   // // TIF[14].SBottom : Werkeug neu: Größe unten / Tool new: size bottom / Herramienta nueva: tamaño abajo
   // // TIF[15].SBottom : Werkeug neu: Größe unten / Tool new: size bottom / Herramienta nueva: tamaño abajo
   // // TIF[16].SBottom : Werkeug neu: Größe unten / Tool new: size bottom / Herramienta nueva: tamaño abajo
   // // TIF[2].TInBuffer : ID für Werkzeuge im Puffer / ID for tools in buffer / ID para herramientas en búfer
   // // TIF[3].TInBuffer : ID für Werkzeuge im Puffer / ID for tools in buffer / ID para herramientas en búfer
   // // TIF[4].TInBuffer : ID für Werkzeuge im Puffer / ID for tools in buffer / ID para herramientas en búfer
   // // TIF[5].TInBuffer : ID für Werkzeuge im Puffer / ID for tools in buffer / ID para herramientas en búfer
   // // TIF[6].TInBuffer : ID für Werkzeuge im Puffer / ID for tools in buffer / ID para herramientas en búfer
   // // TIF[7].TInBuffer : ID für Werkzeuge im Puffer / ID for tools in buffer / ID para herramientas en búfer
   // // TIF[8].TInBuffer : ID für Werkzeuge im Puffer / ID for tools in buffer / ID para herramientas en búfer
   // // TIF[9].TInBuffer : ID für Werkzeuge im Puffer / ID for tools in buffer / ID para herramientas en búfer
   // // TIF[10].TInBuffer : ID für Werkzeuge im Puffer / ID for tools in buffer / ID para herramientas en búfer
   // // TIF[11].TInBuffer : ID für Werkzeuge im Puffer / ID for tools in buffer / ID para herramientas en búfer
   // // TIF[12].TInBuffer : ID für Werkzeuge im Puffer / ID for tools in buffer / ID para herramientas en búfer
   // // TIF[13].TInBuffer : ID für Werkzeuge im Puffer / ID for tools in buffer / ID para herramientas en búfer
   // // TIF[14].TInBuffer : ID für Werkzeuge im Puffer / ID for tools in buffer / ID para herramientas en búfer
   // // TIF[15].TInBuffer : ID für Werkzeuge im Puffer / ID for tools in buffer / ID para herramientas en búfer
   // // TIF[16].TInBuffer : ID für Werkzeuge im Puffer / ID for tools in buffer / ID para herramientas en búfer
   // // TIF[2].IgnoreDisabled : Deaktiviert ignorieren / Ignore disabled / Ignorar desactivado
   // // TIF[3].IgnoreDisabled : Deaktiviert ignorieren / Ignore disabled / Ignorar desactivado
   // // TIF[4].IgnoreDisabled : Deaktiviert ignorieren / Ignore disabled / Ignorar desactivado
   // // TIF[5].IgnoreDisabled : Deaktiviert ignorieren / Ignore disabled / Ignorar desactivado
   // // TIF[6].IgnoreDisabled : Deaktiviert ignorieren / Ignore disabled / Ignorar desactivado
   // // TIF[7].IgnoreDisabled : Deaktiviert ignorieren / Ignore disabled / Ignorar desactivado
   // // TIF[8].IgnoreDisabled : Deaktiviert ignorieren / Ignore disabled / Ignorar desactivado
   // // TIF[9].IgnoreDisabled : Deaktiviert ignorieren / Ignore disabled / Ignorar desactivado
   // // TIF[10].IgnoreDisabled : Deaktiviert ignorieren / Ignore disabled / Ignorar desactivado
   // // TIF[11].IgnoreDisabled : Deaktiviert ignorieren / Ignore disabled / Ignorar desactivado
   // // TIF[12].IgnoreDisabled : Deaktiviert ignorieren / Ignore disabled / Ignorar desactivado
   // // TIF[13].IgnoreDisabled : Deaktiviert ignorieren / Ignore disabled / Ignorar desactivado
   // // TIF[14].IgnoreDisabled : Deaktiviert ignorieren / Ignore disabled / Ignorar desactivado
   // // TIF[15].IgnoreDisabled : Deaktiviert ignorieren / Ignore disabled / Ignorar desactivado
   // // TIF[16].IgnoreDisabled : Deaktiviert ignorieren / Ignore disabled / Ignorar desactivado
   // // TIF[2].Unload : Zu entladen / To be unloaded / Por descargar
   // // TIF[3].Unload : Zu entladen / To be unloaded / Por descargar
   // // TIF[4].Unload : Zu entladen / To be unloaded / Por descargar
   // // TIF[5].Unload : Zu entladen / To be unloaded / Por descargar
   // // TIF[6].Unload : Zu entladen / To be unloaded / Por descargar
   // // TIF[7].Unload : Zu entladen / To be unloaded / Por descargar
   // // TIF[8].Unload : Zu entladen / To be unloaded / Por descargar
   // // TIF[9].Unload : Zu entladen / To be unloaded / Por descargar
   // // TIF[10].Unload : Zu entladen / To be unloaded / Por descargar
   // // TIF[11].Unload : Zu entladen / To be unloaded / Por descargar
   // // TIF[12].Unload : Zu entladen / To be unloaded / Por descargar
   // // TIF[13].Unload : Zu entladen / To be unloaded / Por descargar
   // // TIF[14].Unload : Zu entladen / To be unloaded / Por descargar
   // // TIF[15].Unload : Zu entladen / To be unloaded / Por descargar
   // // TIF[16].Unload : Zu entladen / To be unloaded / Por descargar
   // // TIF[2].Load : Zu laden / To be loaded / Por cargar
   // // TIF[3].Load : Zu laden / To be loaded / Por cargar
   // // TIF[4].Load : Zu laden / To be loaded / Por cargar
   // // TIF[5].Load : Zu laden / To be loaded / Por cargar
   // // TIF[6].Load : Zu laden / To be loaded / Por cargar
   // // TIF[7].Load : Zu laden / To be loaded / Por cargar
   // // TIF[8].Load : Zu laden / To be loaded / Por cargar
   // // TIF[9].Load : Zu laden / To be loaded / Por cargar
   // // TIF[10].Load : Zu laden / To be loaded / Por cargar
   // // TIF[11].Load : Zu laden / To be loaded / Por cargar
   // // TIF[12].Load : Zu laden / To be loaded / Por cargar
   // // TIF[13].Load : Zu laden / To be loaded / Por cargar
   // // TIF[14].Load : Zu laden / To be loaded / Por cargar
   // // TIF[15].Load : Zu laden / To be loaded / Por cargar
   // // TIF[16].Load : Zu laden / To be loaded / Por cargar
   // // TIF[2].MasterTool : Master-Werkzeug / Master tool / Herramienta maestra
   // // TIF[3].MasterTool : Master-Werkzeug / Master tool / Herramienta maestra
   // // TIF[4].MasterTool : Master-Werkzeug / Master tool / Herramienta maestra
   // // TIF[5].MasterTool : Master-Werkzeug / Master tool / Herramienta maestra
   // // TIF[6].MasterTool : Master-Werkzeug / Master tool / Herramienta maestra
   // // TIF[7].MasterTool : Master-Werkzeug / Master tool / Herramienta maestra
   // // TIF[8].MasterTool : Master-Werkzeug / Master tool / Herramienta maestra
   // // TIF[9].MasterTool : Master-Werkzeug / Master tool / Herramienta maestra
   // // TIF[10].MasterTool : Master-Werkzeug / Master tool / Herramienta maestra
   // // TIF[11].MasterTool : Master-Werkzeug / Master tool / Herramienta maestra
   // // TIF[12].MasterTool : Master-Werkzeug / Master tool / Herramienta maestra
   // // TIF[13].MasterTool : Master-Werkzeug / Master tool / Herramienta maestra
   // // TIF[14].MasterTool : Master-Werkzeug / Master tool / Herramienta maestra
   // // TIF[15].MasterTool : Master-Werkzeug / Master tool / Herramienta maestra
   // // TIF[16].MasterTool : Master-Werkzeug / Master tool / Herramienta maestra
   // // TIF[2].n38_5 : Reserviert / Reserved / Reservado
   // // TIF[3].n38_5 : Reserviert / Reserved / Reservado
   // // TIF[4].n38_5 : Reserviert / Reserved / Reservado
   // // TIF[5].n38_5 : Reserviert / Reserved / Reservado
   // // TIF[6].n38_5 : Reserviert / Reserved / Reservado
   // // TIF[7].n38_5 : Reserviert / Reserved / Reservado
   // // TIF[8].n38_5 : Reserviert / Reserved / Reservado
   // // TIF[9].n38_5 : Reserviert / Reserved / Reservado
   // // TIF[10].n38_5 : Reserviert / Reserved / Reservado
   // // TIF[11].n38_5 : Reserviert / Reserved / Reservado
   // // TIF[12].n38_5 : Reserviert / Reserved / Reservado
   // // TIF[13].n38_5 : Reserviert / Reserved / Reservado
   // // TIF[14].n38_5 : Reserviert / Reserved / Reservado
   // // TIF[15].n38_5 : Reserviert / Reserved / Reservado
   // // TIF[16].n38_5 : Reserviert / Reserved / Reservado
   // // TIF[2].Exchange_1to1 : 1:1 Austausch / 1:1 exchange / Cambio 1:1
   // // TIF[3].Exchange_1to1 : 1:1 Austausch / 1:1 exchange / Cambio 1:1
   // // TIF[4].Exchange_1to1 : 1:1 Austausch / 1:1 exchange / Cambio 1:1
   // // TIF[5].Exchange_1to1 : 1:1 Austausch / 1:1 exchange / Cambio 1:1
   // // TIF[6].Exchange_1to1 : 1:1 Austausch / 1:1 exchange / Cambio 1:1
   // // TIF[7].Exchange_1to1 : 1:1 Austausch / 1:1 exchange / Cambio 1:1
   // // TIF[8].Exchange_1to1 : 1:1 Austausch / 1:1 exchange / Cambio 1:1
   // // TIF[9].Exchange_1to1 : 1:1 Austausch / 1:1 exchange / Cambio 1:1
   // // TIF[10].Exchange_1to1 : 1:1 Austausch / 1:1 exchange / Cambio 1:1
   // // TIF[11].Exchange_1to1 : 1:1 Austausch / 1:1 exchange / Cambio 1:1
   // // TIF[12].Exchange_1to1 : 1:1 Austausch / 1:1 exchange / Cambio 1:1
   // // TIF[13].Exchange_1to1 : 1:1 Austausch / 1:1 exchange / Cambio 1:1
   // // TIF[14].Exchange_1to1 : 1:1 Austausch / 1:1 exchange / Cambio 1:1
   // // TIF[15].Exchange_1to1 : 1:1 Austausch / 1:1 exchange / Cambio 1:1
   // // TIF[16].Exchange_1to1 : 1:1 Austausch / 1:1 exchange / Cambio 1:1
   // // TIF[2].HandTool : Handwerkzeug / Hand tool / Herramienta manual
   // // TIF[3].HandTool : Handwerkzeug / Hand tool / Herramienta manual
   // // TIF[4].HandTool : Handwerkzeug / Hand tool / Herramienta manual
   // // TIF[5].HandTool : Handwerkzeug / Hand tool / Herramienta manual
   // // TIF[6].HandTool : Handwerkzeug / Hand tool / Herramienta manual
   // // TIF[7].HandTool : Handwerkzeug / Hand tool / Herramienta manual
   // // TIF[8].HandTool : Handwerkzeug / Hand tool / Herramienta manual
   // // TIF[9].HandTool : Handwerkzeug / Hand tool / Herramienta manual
   // // TIF[10].HandTool : Handwerkzeug / Hand tool / Herramienta manual
   // // TIF[11].HandTool : Handwerkzeug / Hand tool / Herramienta manual
   // // TIF[12].HandTool : Handwerkzeug / Hand tool / Herramienta manual
   // // TIF[13].HandTool : Handwerkzeug / Hand tool / Herramienta manual
   // // TIF[14].HandTool : Handwerkzeug / Hand tool / Herramienta manual
   // // TIF[15].HandTool : Handwerkzeug / Hand tool / Herramienta manual
   // // TIF[16].HandTool : Handwerkzeug / Hand tool / Herramienta manual
   // // TIF[2].Active : Aktives Werkzeug / Active tool / Herramienta activa
   // // TIF[3].Active : Aktives Werkzeug / Active tool / Herramienta activa
   // // TIF[4].Active : Aktives Werkzeug / Active tool / Herramienta activa
   // // TIF[5].Active : Aktives Werkzeug / Active tool / Herramienta activa
   // // TIF[6].Active : Aktives Werkzeug / Active tool / Herramienta activa
   // // TIF[7].Active : Aktives Werkzeug / Active tool / Herramienta activa
   // // TIF[8].Active : Aktives Werkzeug / Active tool / Herramienta activa
   // // TIF[9].Active : Aktives Werkzeug / Active tool / Herramienta activa
   // // TIF[10].Active : Aktives Werkzeug / Active tool / Herramienta activa
   // // TIF[11].Active : Aktives Werkzeug / Active tool / Herramienta activa
   // // TIF[12].Active : Aktives Werkzeug / Active tool / Herramienta activa
   // // TIF[13].Active : Aktives Werkzeug / Active tool / Herramienta activa
   // // TIF[14].Active : Aktives Werkzeug / Active tool / Herramienta activa
   // // TIF[15].Active : Aktives Werkzeug / Active tool / Herramienta activa
   // // TIF[16].Active : Aktives Werkzeug / Active tool / Herramienta activa
   // // TIF[2].Enabled : Werkzeug aktiviert / Tool enabled / Herramienta activada
   // // TIF[3].Enabled : Werkzeug aktiviert / Tool enabled / Herramienta activada
   // // TIF[4].Enabled : Werkzeug aktiviert / Tool enabled / Herramienta activada
   // // TIF[5].Enabled : Werkzeug aktiviert / Tool enabled / Herramienta activada
   // // TIF[6].Enabled : Werkzeug aktiviert / Tool enabled / Herramienta activada
   // // TIF[7].Enabled : Werkzeug aktiviert / Tool enabled / Herramienta activada
   // // TIF[8].Enabled : Werkzeug aktiviert / Tool enabled / Herramienta activada
   // // TIF[9].Enabled : Werkzeug aktiviert / Tool enabled / Herramienta activada
   // // TIF[10].Enabled : Werkzeug aktiviert / Tool enabled / Herramienta activada
   // // TIF[11].Enabled : Werkzeug aktiviert / Tool enabled / Herramienta activada
   // // TIF[12].Enabled : Werkzeug aktiviert / Tool enabled / Herramienta activada
   // // TIF[13].Enabled : Werkzeug aktiviert / Tool enabled / Herramienta activada
   // // TIF[14].Enabled : Werkzeug aktiviert / Tool enabled / Herramienta activada
   // // TIF[15].Enabled : Werkzeug aktiviert / Tool enabled / Herramienta activada
   // // TIF[16].Enabled : Werkzeug aktiviert / Tool enabled / Herramienta activada
   // // TIF[2].Disabled : Werkzeug deaktiviert / Tool disabled / Herramienta desactivada
   // // TIF[3].Disabled : Werkzeug deaktiviert / Tool disabled / Herramienta desactivada
   // // TIF[4].Disabled : Werkzeug deaktiviert / Tool disabled / Herramienta desactivada
   // // TIF[5].Disabled : Werkzeug deaktiviert / Tool disabled / Herramienta desactivada
   // // TIF[6].Disabled : Werkzeug deaktiviert / Tool disabled / Herramienta desactivada
   // // TIF[7].Disabled : Werkzeug deaktiviert / Tool disabled / Herramienta desactivada
   // // TIF[8].Disabled : Werkzeug deaktiviert / Tool disabled / Herramienta desactivada
   // // TIF[9].Disabled : Werkzeug deaktiviert / Tool disabled / Herramienta desactivada
   // // TIF[10].Disabled : Werkzeug deaktiviert / Tool disabled / Herramienta desactivada
   // // TIF[11].Disabled : Werkzeug deaktiviert / Tool disabled / Herramienta desactivada
   // // TIF[12].Disabled : Werkzeug deaktiviert / Tool disabled / Herramienta desactivada
   // // TIF[13].Disabled : Werkzeug deaktiviert / Tool disabled / Herramienta desactivada
   // // TIF[14].Disabled : Werkzeug deaktiviert / Tool disabled / Herramienta desactivada
   // // TIF[15].Disabled : Werkzeug deaktiviert / Tool disabled / Herramienta desactivada
   // // TIF[16].Disabled : Werkzeug deaktiviert / Tool disabled / Herramienta desactivada
   // // TIF[2].Measured : Werkzeug gemessen / Tool measured / Herramienta medida
   // // TIF[3].Measured : Werkzeug gemessen / Tool measured / Herramienta medida
   // // TIF[4].Measured : Werkzeug gemessen / Tool measured / Herramienta medida
   // // TIF[5].Measured : Werkzeug gemessen / Tool measured / Herramienta medida
   // // TIF[6].Measured : Werkzeug gemessen / Tool measured / Herramienta medida
   // // TIF[7].Measured : Werkzeug gemessen / Tool measured / Herramienta medida
   // // TIF[8].Measured : Werkzeug gemessen / Tool measured / Herramienta medida
   // // TIF[9].Measured : Werkzeug gemessen / Tool measured / Herramienta medida
   // // TIF[10].Measured : Werkzeug gemessen / Tool measured / Herramienta medida
   // // TIF[11].Measured : Werkzeug gemessen / Tool measured / Herramienta medida
   // // TIF[12].Measured : Werkzeug gemessen / Tool measured / Herramienta medida
   // // TIF[13].Measured : Werkzeug gemessen / Tool measured / Herramienta medida
   // // TIF[14].Measured : Werkzeug gemessen / Tool measured / Herramienta medida
   // // TIF[15].Measured : Werkzeug gemessen / Tool measured / Herramienta medida
   // // TIF[16].Measured : Werkzeug gemessen / Tool measured / Herramienta medida
   // // TIF[2].Prewarn : Vorwarnungsgrenze erreicht / Prewarning limit reached / Límite de prealarma alcanzado
   // // TIF[3].Prewarn : Vorwarnungsgrenze erreicht / Prewarning limit reached / Límite de prealarma alcanzado
   // // TIF[4].Prewarn : Vorwarnungsgrenze erreicht / Prewarning limit reached / Límite de prealarma alcanzado
   // // TIF[5].Prewarn : Vorwarnungsgrenze erreicht / Prewarning limit reached / Límite de prealarma alcanzado
   // // TIF[6].Prewarn : Vorwarnungsgrenze erreicht / Prewarning limit reached / Límite de prealarma alcanzado
   // // TIF[7].Prewarn : Vorwarnungsgrenze erreicht / Prewarning limit reached / Límite de prealarma alcanzado
   // // TIF[8].Prewarn : Vorwarnungsgrenze erreicht / Prewarning limit reached / Límite de prealarma alcanzado
   // // TIF[9].Prewarn : Vorwarnungsgrenze erreicht / Prewarning limit reached / Límite de prealarma alcanzado
   // // TIF[10].Prewarn : Vorwarnungsgrenze erreicht / Prewarning limit reached / Límite de prealarma alcanzado
   // // TIF[11].Prewarn : Vorwarnungsgrenze erreicht / Prewarning limit reached / Límite de prealarma alcanzado
   // // TIF[12].Prewarn : Vorwarnungsgrenze erreicht / Prewarning limit reached / Límite de prealarma alcanzado
   // // TIF[13].Prewarn : Vorwarnungsgrenze erreicht / Prewarning limit reached / Límite de prealarma alcanzado
   // // TIF[14].Prewarn : Vorwarnungsgrenze erreicht / Prewarning limit reached / Límite de prealarma alcanzado
   // // TIF[15].Prewarn : Vorwarnungsgrenze erreicht / Prewarning limit reached / Límite de prealarma alcanzado
   // // TIF[16].Prewarn : Vorwarnungsgrenze erreicht / Prewarning limit reached / Límite de prealarma alcanzado
   // // TIF[2].Change : Werkzeug wird gewechselt / Tool being changed / Sustituyendo herramienta
   // // TIF[3].Change : Werkzeug wird gewechselt / Tool being changed / Sustituyendo herramienta
   // // TIF[4].Change : Werkzeug wird gewechselt / Tool being changed / Sustituyendo herramienta
   // // TIF[5].Change : Werkzeug wird gewechselt / Tool being changed / Sustituyendo herramienta
   // // TIF[6].Change : Werkzeug wird gewechselt / Tool being changed / Sustituyendo herramienta
   // // TIF[7].Change : Werkzeug wird gewechselt / Tool being changed / Sustituyendo herramienta
   // // TIF[8].Change : Werkzeug wird gewechselt / Tool being changed / Sustituyendo herramienta
   // // TIF[9].Change : Werkzeug wird gewechselt / Tool being changed / Sustituyendo herramienta
   // // TIF[10].Change : Werkzeug wird gewechselt / Tool being changed / Sustituyendo herramienta
   // // TIF[11].Change : Werkzeug wird gewechselt / Tool being changed / Sustituyendo herramienta
   // // TIF[12].Change : Werkzeug wird gewechselt / Tool being changed / Sustituyendo herramienta
   // // TIF[13].Change : Werkzeug wird gewechselt / Tool being changed / Sustituyendo herramienta
   // // TIF[14].Change : Werkzeug wird gewechselt / Tool being changed / Sustituyendo herramienta
   // // TIF[15].Change : Werkzeug wird gewechselt / Tool being changed / Sustituyendo herramienta
   // // TIF[16].Change : Werkzeug wird gewechselt / Tool being changed / Sustituyendo herramienta
   // // TIF[2].FixedLoc : Werkzeug-Festplatz codiert / Tool fixed location coded / Puesto fijo de herramienta codificado
   // // TIF[3].FixedLoc : Werkzeug-Festplatz codiert / Tool fixed location coded / Puesto fijo de herramienta codificado
   // // TIF[4].FixedLoc : Werkzeug-Festplatz codiert / Tool fixed location coded / Puesto fijo de herramienta codificado
   // // TIF[5].FixedLoc : Werkzeug-Festplatz codiert / Tool fixed location coded / Puesto fijo de herramienta codificado
   // // TIF[6].FixedLoc : Werkzeug-Festplatz codiert / Tool fixed location coded / Puesto fijo de herramienta codificado
   // // TIF[7].FixedLoc : Werkzeug-Festplatz codiert / Tool fixed location coded / Puesto fijo de herramienta codificado
   // // TIF[8].FixedLoc : Werkzeug-Festplatz codiert / Tool fixed location coded / Puesto fijo de herramienta codificado
   // // TIF[9].FixedLoc : Werkzeug-Festplatz codiert / Tool fixed location coded / Puesto fijo de herramienta codificado
   // // TIF[10].FixedLoc : Werkzeug-Festplatz codiert / Tool fixed location coded / Puesto fijo de herramienta codificado
   // // TIF[11].FixedLoc : Werkzeug-Festplatz codiert / Tool fixed location coded / Puesto fijo de herramienta codificado
   // // TIF[12].FixedLoc : Werkzeug-Festplatz codiert / Tool fixed location coded / Puesto fijo de herramienta codificado
   // // TIF[13].FixedLoc : Werkzeug-Festplatz codiert / Tool fixed location coded / Puesto fijo de herramienta codificado
   // // TIF[14].FixedLoc : Werkzeug-Festplatz codiert / Tool fixed location coded / Puesto fijo de herramienta codificado
   // // TIF[15].FixedLoc : Werkzeug-Festplatz codiert / Tool fixed location coded / Puesto fijo de herramienta codificado
   // // TIF[16].FixedLoc : Werkzeug-Festplatz codiert / Tool fixed location coded / Puesto fijo de herramienta codificado
   // // TIF[2].Used : Werkzeug war in Gebrauch / Tool was in use / La herramienta estaba en uso
   // // TIF[3].Used : Werkzeug war in Gebrauch / Tool was in use / La herramienta estaba en uso
   // // TIF[4].Used : Werkzeug war in Gebrauch / Tool was in use / La herramienta estaba en uso
   // // TIF[5].Used : Werkzeug war in Gebrauch / Tool was in use / La herramienta estaba en uso
   // // TIF[6].Used : Werkzeug war in Gebrauch / Tool was in use / La herramienta estaba en uso
   // // TIF[7].Used : Werkzeug war in Gebrauch / Tool was in use / La herramienta estaba en uso
   // // TIF[8].Used : Werkzeug war in Gebrauch / Tool was in use / La herramienta estaba en uso
   // // TIF[9].Used : Werkzeug war in Gebrauch / Tool was in use / La herramienta estaba en uso
   // // TIF[10].Used : Werkzeug war in Gebrauch / Tool was in use / La herramienta estaba en uso
   // // TIF[11].Used : Werkzeug war in Gebrauch / Tool was in use / La herramienta estaba en uso
   // // TIF[12].Used : Werkzeug war in Gebrauch / Tool was in use / La herramienta estaba en uso
   // // TIF[13].Used : Werkzeug war in Gebrauch / Tool was in use / La herramienta estaba en uso
   // // TIF[14].Used : Werkzeug war in Gebrauch / Tool was in use / La herramienta estaba en uso
   // // TIF[15].Used : Werkzeug war in Gebrauch / Tool was in use / La herramienta estaba en uso
   // // TIF[16].Used : Werkzeug war in Gebrauch / Tool was in use / La herramienta estaba en uso
   // // TIF[2].TNo : Werkzeug neu: WZ-Nummer / Tool new: T number / Herramienta nueva: n.º herramienta
   // // TIF[3].TNo : Werkzeug neu: WZ-Nummer / Tool new: T number / Herramienta nueva: n.º herramienta
   // // TIF[4].TNo : Werkzeug neu: WZ-Nummer / Tool new: T number / Herramienta nueva: n.º herramienta
   // // TIF[5].TNo : Werkzeug neu: WZ-Nummer / Tool new: T number / Herramienta nueva: n.º herramienta
   // // TIF[6].TNo : Werkzeug neu: WZ-Nummer / Tool new: T number / Herramienta nueva: n.º herramienta
   // // TIF[7].TNo : Werkzeug neu: WZ-Nummer / Tool new: T number / Herramienta nueva: n.º herramienta
   // // TIF[8].TNo : Werkzeug neu: WZ-Nummer / Tool new: T number / Herramienta nueva: n.º herramienta
   // // TIF[9].TNo : Werkzeug neu: WZ-Nummer / Tool new: T number / Herramienta nueva: n.º herramienta
   // // TIF[10].TNo : Werkzeug neu: WZ-Nummer / Tool new: T number / Herramienta nueva: n.º herramienta
   // // TIF[11].TNo : Werkzeug neu: WZ-Nummer / Tool new: T number / Herramienta nueva: n.º herramienta
   // // TIF[12].TNo : Werkzeug neu: WZ-Nummer / Tool new: T number / Herramienta nueva: n.º herramienta
   // // TIF[13].TNo : Werkzeug neu: WZ-Nummer / Tool new: T number / Herramienta nueva: n.º herramienta
   // // TIF[14].TNo : Werkzeug neu: WZ-Nummer / Tool new: T number / Herramienta nueva: n.º herramienta
   // // TIF[15].TNo : Werkzeug neu: WZ-Nummer / Tool new: T number / Herramienta nueva: n.º herramienta
   // // TIF[16].TNo : Werkzeug neu: WZ-Nummer / Tool new: T number / Herramienta nueva: n.º herramienta
   // // TIF[2].OldTBufferNo : Puffernummer des vorherigen Werkzeugs / Buffer number of previous tool / Número de búfer de la herramienta previa
   // // TIF[3].OldTBufferNo : Puffernummer des vorherigen Werkzeugs / Buffer number of previous tool / Número de búfer de la herramienta previa
   // // TIF[4].OldTBufferNo : Puffernummer des vorherigen Werkzeugs / Buffer number of previous tool / Número de búfer de la herramienta previa
   // // TIF[5].OldTBufferNo : Puffernummer des vorherigen Werkzeugs / Buffer number of previous tool / Número de búfer de la herramienta previa
   // // TIF[6].OldTBufferNo : Puffernummer des vorherigen Werkzeugs / Buffer number of previous tool / Número de búfer de la herramienta previa
   // // TIF[7].OldTBufferNo : Puffernummer des vorherigen Werkzeugs / Buffer number of previous tool / Número de búfer de la herramienta previa
   // // TIF[8].OldTBufferNo : Puffernummer des vorherigen Werkzeugs / Buffer number of previous tool / Número de búfer de la herramienta previa
   // // TIF[9].OldTBufferNo : Puffernummer des vorherigen Werkzeugs / Buffer number of previous tool / Número de búfer de la herramienta previa
   // // TIF[10].OldTBufferNo : Puffernummer des vorherigen Werkzeugs / Buffer number of previous tool / Número de búfer de la herramienta previa
   // // TIF[11].OldTBufferNo : Puffernummer des vorherigen Werkzeugs / Buffer number of previous tool / Número de búfer de la herramienta previa
   // // TIF[12].OldTBufferNo : Puffernummer des vorherigen Werkzeugs / Buffer number of previous tool / Número de búfer de la herramienta previa
   // // TIF[13].OldTBufferNo : Puffernummer des vorherigen Werkzeugs / Buffer number of previous tool / Número de búfer de la herramienta previa
   // // TIF[14].OldTBufferNo : Puffernummer des vorherigen Werkzeugs / Buffer number of previous tool / Número de búfer de la herramienta previa
   // // TIF[15].OldTBufferNo : Puffernummer des vorherigen Werkzeugs / Buffer number of previous tool / Número de búfer de la herramienta previa
   // // TIF[16].OldTBufferNo : Puffernummer des vorherigen Werkzeugs / Buffer number of previous tool / Número de búfer de la herramienta previa
   // // TIF[2].MyMag : Originalmagazin des neuen Werkzeugs / Original magazine of new tool / Almacén de origen de la nueva herramienta
   // // TIF[3].MyMag : Originalmagazin des neuen Werkzeugs / Original magazine of new tool / Almacén de origen de la nueva herramienta
   // // TIF[4].MyMag : Originalmagazin des neuen Werkzeugs / Original magazine of new tool / Almacén de origen de la nueva herramienta
   // // TIF[5].MyMag : Originalmagazin des neuen Werkzeugs / Original magazine of new tool / Almacén de origen de la nueva herramienta
   // // TIF[6].MyMag : Originalmagazin des neuen Werkzeugs / Original magazine of new tool / Almacén de origen de la nueva herramienta
   // // TIF[7].MyMag : Originalmagazin des neuen Werkzeugs / Original magazine of new tool / Almacén de origen de la nueva herramienta
   // // TIF[8].MyMag : Originalmagazin des neuen Werkzeugs / Original magazine of new tool / Almacén de origen de la nueva herramienta
   // // TIF[9].MyMag : Originalmagazin des neuen Werkzeugs / Original magazine of new tool / Almacén de origen de la nueva herramienta
   // // TIF[10].MyMag : Originalmagazin des neuen Werkzeugs / Original magazine of new tool / Almacén de origen de la nueva herramienta
   // // TIF[11].MyMag : Originalmagazin des neuen Werkzeugs / Original magazine of new tool / Almacén de origen de la nueva herramienta
   // // TIF[12].MyMag : Originalmagazin des neuen Werkzeugs / Original magazine of new tool / Almacén de origen de la nueva herramienta
   // // TIF[13].MyMag : Originalmagazin des neuen Werkzeugs / Original magazine of new tool / Almacén de origen de la nueva herramienta
   // // TIF[14].MyMag : Originalmagazin des neuen Werkzeugs / Original magazine of new tool / Almacén de origen de la nueva herramienta
   // // TIF[15].MyMag : Originalmagazin des neuen Werkzeugs / Original magazine of new tool / Almacén de origen de la nueva herramienta
   // // TIF[16].MyMag : Originalmagazin des neuen Werkzeugs / Original magazine of new tool / Almacén de origen de la nueva herramienta
   // // TIF[2].MyPlace : Originalplatz des neuen Werkzeugs / Original location of new tool / Puesto de origen de la nueva herramienta
   // // TIF[3].MyPlace : Originalplatz des neuen Werkzeugs / Original location of new tool / Puesto de origen de la nueva herramienta
   // // TIF[4].MyPlace : Originalplatz des neuen Werkzeugs / Original location of new tool / Puesto de origen de la nueva herramienta
   // // TIF[5].MyPlace : Originalplatz des neuen Werkzeugs / Original location of new tool / Puesto de origen de la nueva herramienta
   // // TIF[6].MyPlace : Originalplatz des neuen Werkzeugs / Original location of new tool / Puesto de origen de la nueva herramienta
   // // TIF[7].MyPlace : Originalplatz des neuen Werkzeugs / Original location of new tool / Puesto de origen de la nueva herramienta
   // // TIF[8].MyPlace : Originalplatz des neuen Werkzeugs / Original location of new tool / Puesto de origen de la nueva herramienta
   // // TIF[9].MyPlace : Originalplatz des neuen Werkzeugs / Original location of new tool / Puesto de origen de la nueva herramienta
   // // TIF[10].MyPlace : Originalplatz des neuen Werkzeugs / Original location of new tool / Puesto de origen de la nueva herramienta
   // // TIF[11].MyPlace : Originalplatz des neuen Werkzeugs / Original location of new tool / Puesto de origen de la nueva herramienta
   // // TIF[12].MyPlace : Originalplatz des neuen Werkzeugs / Original location of new tool / Puesto de origen de la nueva herramienta
   // // TIF[13].MyPlace : Originalplatz des neuen Werkzeugs / Original location of new tool / Puesto de origen de la nueva herramienta
   // // TIF[14].MyPlace : Originalplatz des neuen Werkzeugs / Original location of new tool / Puesto de origen de la nueva herramienta
   // // TIF[15].MyPlace : Originalplatz des neuen Werkzeugs / Original location of new tool / Puesto de origen de la nueva herramienta
   // // TIF[16].MyPlace : Originalplatz des neuen Werkzeugs / Original location of new tool / Puesto de origen de la nueva herramienta
END_TYPE

TYPE "LBP_typeTMSpindleMT"
TITLE = Tool management / Gestión de herramientas / Werkzeugverwaltung
// User data type for block LBP_TMSpindleMT [DB1072] / Tipo de dato de usuario para bloque LBP_TMSpindleMT [DB1072] / Anwender-Datentyp für Baustein LBP_TMSpindleMT [DB1072]
// stored: IsFailsafeCompliant false
   STRUCT
      MTIF : Array[1..16] of Struct
         DistanceCoding : Int;   // Art der Entfernungscodierung ($TC_MTP_KD) / Type of distance coding ($TC_MTP_KD) / Tipo de codificación de distancia ($TC_MTP_KD)
         Places : Int;   // Anzahl der Plätze des Multitools / Number of locations of the multitool / Número de puestos de Multitool
         Distance : Real;   // Entfernung des Multitool-Platzes / Multitool location distance / Distancia a puesto Multitool
         NewMTNo : Int;   // MT-Nummer des neuen Tools / MT number of new tool / Número MT de la nueva herramienta
         NewPlace : Int;   // Multitool-Platznummer / Multitool place number / Número de puesto de Multitool
         OldMTNo : Int;   // MT-Nummer des vorherigen Tools / MT number of previous tool / Número MT de la herramienta previa
         OldPlace : Int;   // Multitool-Platznummer / Multitool place number / Número de puesto de Multitool
         LocType : Int;   // Werkzeug neu: Platzart / Tool new: location type / Herramienta nueva: tipo de puesto
         SLeft : Int;   // Werkeug neu: Größe links / Tool new: size left / Herramienta nueva: tamaño izquierda
         SRight : Int;   // Werkeug neu: Größe rechts / Tool new: size right / Herramienta nueva: tamaño derecha
         STop : Int;   // Werkeug neu: Größe oben / Tool new: size top / Herramienta nueva: tamaño arriba
         SBottom : Int;   // Werkeug neu: Größe unten / Tool new: size bottom / Herramienta nueva: tamaño abajo
         TInBuffer : Bool;   // ID für Werkzeuge im Puffer / ID for tools in buffer / ID para herramientas en búfer
         IgnoreDisabled : Bool;   // Deaktiviert ignorieren / Ignore disabled / Ignorar desactivado
         Unload : Bool;   // Zu entladen / To be unloaded / Por descargar
         Load : Bool;   // Zu laden / To be loaded / Por cargar
         MasterTool : Bool;   // Master-Werkzeug / Master tool / Herramienta maestra
         n26_5 : Bool;   // Reserviert / Reserved / Reservado
         n26_6 : Bool;   // Reserviert / Reserved / Reservado
         HandTool : Bool;   // Handwerkzeug / Hand tool / Herramienta manual
         Active : Bool;   // Aktives Werkzeug / Active tool / Herramienta activa
         Enabled : Bool;   // Werkzeug aktiviert / Tool enabled / Herramienta activada
         Disabled : Bool;   // Werkzeug deaktiviert / Tool disabled / Herramienta desactivada
         Measured : Bool;   // Werkzeug gemessen / Tool measured / Herramienta medida
         Prewarn : Bool;   // Vorwarnungsgrenze erreicht / Prewarning limit reached / Límite de prealarma alcanzado
         Change : Bool;   // Werkzeug wird gewechselt / Tool being changed / Sustituyendo herramienta
         FixedLoc : Bool;   // Werkzeug-Festplatz codiert / Tool fixed location coded / Puesto fijo de herramienta codificado
         Used : Bool;   // Werkzeug war in Gebrauch / Tool was in use / La herramienta estaba en uso
         TNo : Int;   // Werkzeug neu: WZ-Nummer / Tool new: T number / Herramienta nueva: n.º herramienta
         Toolholder : Int;   // Werkzeughalter-Nummer als Referenz für die Werkzeugkompensation / Toolholder number as tool compensation reference / Número de portaherramientas como referencia para compensación de herramientas
         MyMag : Int;   // Multitool-Nummer, in die das Werkzeug geladen wird / Multitool number the tool is loaded onto / Número de Multitool en el que se carga la herramienta
         MyPlace : Int;   // Multitool-Platznummer / Multitool place number / Número de puesto de Multitool
         reserved : Array[1..7] of Int;   // Reserviert / Reserved / Reservado
      END_STRUCT;
   END_STRUCT;
   // // MTIF[2].DistanceCoding : Art der Entfernungscodierung ($TC_MTP_KD) / Type of distance coding ($TC_MTP_KD) / Tipo de codificación de distancia ($TC_MTP_KD)
   // // MTIF[3].DistanceCoding : Art der Entfernungscodierung ($TC_MTP_KD) / Type of distance coding ($TC_MTP_KD) / Tipo de codificación de distancia ($TC_MTP_KD)
   // // MTIF[4].DistanceCoding : Art der Entfernungscodierung ($TC_MTP_KD) / Type of distance coding ($TC_MTP_KD) / Tipo de codificación de distancia ($TC_MTP_KD)
   // // MTIF[5].DistanceCoding : Art der Entfernungscodierung ($TC_MTP_KD) / Type of distance coding ($TC_MTP_KD) / Tipo de codificación de distancia ($TC_MTP_KD)
   // // MTIF[6].DistanceCoding : Art der Entfernungscodierung ($TC_MTP_KD) / Type of distance coding ($TC_MTP_KD) / Tipo de codificación de distancia ($TC_MTP_KD)
   // // MTIF[7].DistanceCoding : Art der Entfernungscodierung ($TC_MTP_KD) / Type of distance coding ($TC_MTP_KD) / Tipo de codificación de distancia ($TC_MTP_KD)
   // // MTIF[8].DistanceCoding : Art der Entfernungscodierung ($TC_MTP_KD) / Type of distance coding ($TC_MTP_KD) / Tipo de codificación de distancia ($TC_MTP_KD)
   // // MTIF[9].DistanceCoding : Art der Entfernungscodierung ($TC_MTP_KD) / Type of distance coding ($TC_MTP_KD) / Tipo de codificación de distancia ($TC_MTP_KD)
   // // MTIF[10].DistanceCoding : Art der Entfernungscodierung ($TC_MTP_KD) / Type of distance coding ($TC_MTP_KD) / Tipo de codificación de distancia ($TC_MTP_KD)
   // // MTIF[11].DistanceCoding : Art der Entfernungscodierung ($TC_MTP_KD) / Type of distance coding ($TC_MTP_KD) / Tipo de codificación de distancia ($TC_MTP_KD)
   // // MTIF[12].DistanceCoding : Art der Entfernungscodierung ($TC_MTP_KD) / Type of distance coding ($TC_MTP_KD) / Tipo de codificación de distancia ($TC_MTP_KD)
   // // MTIF[13].DistanceCoding : Art der Entfernungscodierung ($TC_MTP_KD) / Type of distance coding ($TC_MTP_KD) / Tipo de codificación de distancia ($TC_MTP_KD)
   // // MTIF[14].DistanceCoding : Art der Entfernungscodierung ($TC_MTP_KD) / Type of distance coding ($TC_MTP_KD) / Tipo de codificación de distancia ($TC_MTP_KD)
   // // MTIF[15].DistanceCoding : Art der Entfernungscodierung ($TC_MTP_KD) / Type of distance coding ($TC_MTP_KD) / Tipo de codificación de distancia ($TC_MTP_KD)
   // // MTIF[16].DistanceCoding : Art der Entfernungscodierung ($TC_MTP_KD) / Type of distance coding ($TC_MTP_KD) / Tipo de codificación de distancia ($TC_MTP_KD)
   // // MTIF[2].Places : Anzahl der Plätze des Multitools / Number of locations of the multitool / Número de puestos de Multitool
   // // MTIF[3].Places : Anzahl der Plätze des Multitools / Number of locations of the multitool / Número de puestos de Multitool
   // // MTIF[4].Places : Anzahl der Plätze des Multitools / Number of locations of the multitool / Número de puestos de Multitool
   // // MTIF[5].Places : Anzahl der Plätze des Multitools / Number of locations of the multitool / Número de puestos de Multitool
   // // MTIF[6].Places : Anzahl der Plätze des Multitools / Number of locations of the multitool / Número de puestos de Multitool
   // // MTIF[7].Places : Anzahl der Plätze des Multitools / Number of locations of the multitool / Número de puestos de Multitool
   // // MTIF[8].Places : Anzahl der Plätze des Multitools / Number of locations of the multitool / Número de puestos de Multitool
   // // MTIF[9].Places : Anzahl der Plätze des Multitools / Number of locations of the multitool / Número de puestos de Multitool
   // // MTIF[10].Places : Anzahl der Plätze des Multitools / Number of locations of the multitool / Número de puestos de Multitool
   // // MTIF[11].Places : Anzahl der Plätze des Multitools / Number of locations of the multitool / Número de puestos de Multitool
   // // MTIF[12].Places : Anzahl der Plätze des Multitools / Number of locations of the multitool / Número de puestos de Multitool
   // // MTIF[13].Places : Anzahl der Plätze des Multitools / Number of locations of the multitool / Número de puestos de Multitool
   // // MTIF[14].Places : Anzahl der Plätze des Multitools / Number of locations of the multitool / Número de puestos de Multitool
   // // MTIF[15].Places : Anzahl der Plätze des Multitools / Number of locations of the multitool / Número de puestos de Multitool
   // // MTIF[16].Places : Anzahl der Plätze des Multitools / Number of locations of the multitool / Número de puestos de Multitool
   // // MTIF[2].Distance : Entfernung des Multitool-Platzes / Multitool location distance / Distancia a puesto Multitool
   // // MTIF[3].Distance : Entfernung des Multitool-Platzes / Multitool location distance / Distancia a puesto Multitool
   // // MTIF[4].Distance : Entfernung des Multitool-Platzes / Multitool location distance / Distancia a puesto Multitool
   // // MTIF[5].Distance : Entfernung des Multitool-Platzes / Multitool location distance / Distancia a puesto Multitool
   // // MTIF[6].Distance : Entfernung des Multitool-Platzes / Multitool location distance / Distancia a puesto Multitool
   // // MTIF[7].Distance : Entfernung des Multitool-Platzes / Multitool location distance / Distancia a puesto Multitool
   // // MTIF[8].Distance : Entfernung des Multitool-Platzes / Multitool location distance / Distancia a puesto Multitool
   // // MTIF[9].Distance : Entfernung des Multitool-Platzes / Multitool location distance / Distancia a puesto Multitool
   // // MTIF[10].Distance : Entfernung des Multitool-Platzes / Multitool location distance / Distancia a puesto Multitool
   // // MTIF[11].Distance : Entfernung des Multitool-Platzes / Multitool location distance / Distancia a puesto Multitool
   // // MTIF[12].Distance : Entfernung des Multitool-Platzes / Multitool location distance / Distancia a puesto Multitool
   // // MTIF[13].Distance : Entfernung des Multitool-Platzes / Multitool location distance / Distancia a puesto Multitool
   // // MTIF[14].Distance : Entfernung des Multitool-Platzes / Multitool location distance / Distancia a puesto Multitool
   // // MTIF[15].Distance : Entfernung des Multitool-Platzes / Multitool location distance / Distancia a puesto Multitool
   // // MTIF[16].Distance : Entfernung des Multitool-Platzes / Multitool location distance / Distancia a puesto Multitool
   // // MTIF[2].NewMTNo : MT-Nummer des neuen Tools / MT number of new tool / Número MT de la nueva herramienta
   // // MTIF[3].NewMTNo : MT-Nummer des neuen Tools / MT number of new tool / Número MT de la nueva herramienta
   // // MTIF[4].NewMTNo : MT-Nummer des neuen Tools / MT number of new tool / Número MT de la nueva herramienta
   // // MTIF[5].NewMTNo : MT-Nummer des neuen Tools / MT number of new tool / Número MT de la nueva herramienta
   // // MTIF[6].NewMTNo : MT-Nummer des neuen Tools / MT number of new tool / Número MT de la nueva herramienta
   // // MTIF[7].NewMTNo : MT-Nummer des neuen Tools / MT number of new tool / Número MT de la nueva herramienta
   // // MTIF[8].NewMTNo : MT-Nummer des neuen Tools / MT number of new tool / Número MT de la nueva herramienta
   // // MTIF[9].NewMTNo : MT-Nummer des neuen Tools / MT number of new tool / Número MT de la nueva herramienta
   // // MTIF[10].NewMTNo : MT-Nummer des neuen Tools / MT number of new tool / Número MT de la nueva herramienta
   // // MTIF[11].NewMTNo : MT-Nummer des neuen Tools / MT number of new tool / Número MT de la nueva herramienta
   // // MTIF[12].NewMTNo : MT-Nummer des neuen Tools / MT number of new tool / Número MT de la nueva herramienta
   // // MTIF[13].NewMTNo : MT-Nummer des neuen Tools / MT number of new tool / Número MT de la nueva herramienta
   // // MTIF[14].NewMTNo : MT-Nummer des neuen Tools / MT number of new tool / Número MT de la nueva herramienta
   // // MTIF[15].NewMTNo : MT-Nummer des neuen Tools / MT number of new tool / Número MT de la nueva herramienta
   // // MTIF[16].NewMTNo : MT-Nummer des neuen Tools / MT number of new tool / Número MT de la nueva herramienta
   // // MTIF[2].NewPlace : Multitool-Platznummer / Multitool place number / Número de puesto de Multitool
   // // MTIF[3].NewPlace : Multitool-Platznummer / Multitool place number / Número de puesto de Multitool
   // // MTIF[4].NewPlace : Multitool-Platznummer / Multitool place number / Número de puesto de Multitool
   // // MTIF[5].NewPlace : Multitool-Platznummer / Multitool place number / Número de puesto de Multitool
   // // MTIF[6].NewPlace : Multitool-Platznummer / Multitool place number / Número de puesto de Multitool
   // // MTIF[7].NewPlace : Multitool-Platznummer / Multitool place number / Número de puesto de Multitool
   // // MTIF[8].NewPlace : Multitool-Platznummer / Multitool place number / Número de puesto de Multitool
   // // MTIF[9].NewPlace : Multitool-Platznummer / Multitool place number / Número de puesto de Multitool
   // // MTIF[10].NewPlace : Multitool-Platznummer / Multitool place number / Número de puesto de Multitool
   // // MTIF[11].NewPlace : Multitool-Platznummer / Multitool place number / Número de puesto de Multitool
   // // MTIF[12].NewPlace : Multitool-Platznummer / Multitool place number / Número de puesto de Multitool
   // // MTIF[13].NewPlace : Multitool-Platznummer / Multitool place number / Número de puesto de Multitool
   // // MTIF[14].NewPlace : Multitool-Platznummer / Multitool place number / Número de puesto de Multitool
   // // MTIF[15].NewPlace : Multitool-Platznummer / Multitool place number / Número de puesto de Multitool
   // // MTIF[16].NewPlace : Multitool-Platznummer / Multitool place number / Número de puesto de Multitool
   // // MTIF[2].OldMTNo : MT-Nummer des vorherigen Tools / MT number of previous tool / Número MT de la herramienta previa
   // // MTIF[3].OldMTNo : MT-Nummer des vorherigen Tools / MT number of previous tool / Número MT de la herramienta previa
   // // MTIF[4].OldMTNo : MT-Nummer des vorherigen Tools / MT number of previous tool / Número MT de la herramienta previa
   // // MTIF[5].OldMTNo : MT-Nummer des vorherigen Tools / MT number of previous tool / Número MT de la herramienta previa
   // // MTIF[6].OldMTNo : MT-Nummer des vorherigen Tools / MT number of previous tool / Número MT de la herramienta previa
   // // MTIF[7].OldMTNo : MT-Nummer des vorherigen Tools / MT number of previous tool / Número MT de la herramienta previa
   // // MTIF[8].OldMTNo : MT-Nummer des vorherigen Tools / MT number of previous tool / Número MT de la herramienta previa
   // // MTIF[9].OldMTNo : MT-Nummer des vorherigen Tools / MT number of previous tool / Número MT de la herramienta previa
   // // MTIF[10].OldMTNo : MT-Nummer des vorherigen Tools / MT number of previous tool / Número MT de la herramienta previa
   // // MTIF[11].OldMTNo : MT-Nummer des vorherigen Tools / MT number of previous tool / Número MT de la herramienta previa
   // // MTIF[12].OldMTNo : MT-Nummer des vorherigen Tools / MT number of previous tool / Número MT de la herramienta previa
   // // MTIF[13].OldMTNo : MT-Nummer des vorherigen Tools / MT number of previous tool / Número MT de la herramienta previa
   // // MTIF[14].OldMTNo : MT-Nummer des vorherigen Tools / MT number of previous tool / Número MT de la herramienta previa
   // // MTIF[15].OldMTNo : MT-Nummer des vorherigen Tools / MT number of previous tool / Número MT de la herramienta previa
   // // MTIF[16].OldMTNo : MT-Nummer des vorherigen Tools / MT number of previous tool / Número MT de la herramienta previa
   // // MTIF[2].OldPlace : Multitool-Platznummer / Multitool place number / Número de puesto de Multitool
   // // MTIF[3].OldPlace : Multitool-Platznummer / Multitool place number / Número de puesto de Multitool
   // // MTIF[4].OldPlace : Multitool-Platznummer / Multitool place number / Número de puesto de Multitool
   // // MTIF[5].OldPlace : Multitool-Platznummer / Multitool place number / Número de puesto de Multitool
   // // MTIF[6].OldPlace : Multitool-Platznummer / Multitool place number / Número de puesto de Multitool
   // // MTIF[7].OldPlace : Multitool-Platznummer / Multitool place number / Número de puesto de Multitool
   // // MTIF[8].OldPlace : Multitool-Platznummer / Multitool place number / Número de puesto de Multitool
   // // MTIF[9].OldPlace : Multitool-Platznummer / Multitool place number / Número de puesto de Multitool
   // // MTIF[10].OldPlace : Multitool-Platznummer / Multitool place number / Número de puesto de Multitool
   // // MTIF[11].OldPlace : Multitool-Platznummer / Multitool place number / Número de puesto de Multitool
   // // MTIF[12].OldPlace : Multitool-Platznummer / Multitool place number / Número de puesto de Multitool
   // // MTIF[13].OldPlace : Multitool-Platznummer / Multitool place number / Número de puesto de Multitool
   // // MTIF[14].OldPlace : Multitool-Platznummer / Multitool place number / Número de puesto de Multitool
   // // MTIF[15].OldPlace : Multitool-Platznummer / Multitool place number / Número de puesto de Multitool
   // // MTIF[16].OldPlace : Multitool-Platznummer / Multitool place number / Número de puesto de Multitool
   // // MTIF[2].LocType : Werkzeug neu: Platzart / Tool new: location type / Herramienta nueva: tipo de puesto
   // // MTIF[3].LocType : Werkzeug neu: Platzart / Tool new: location type / Herramienta nueva: tipo de puesto
   // // MTIF[4].LocType : Werkzeug neu: Platzart / Tool new: location type / Herramienta nueva: tipo de puesto
   // // MTIF[5].LocType : Werkzeug neu: Platzart / Tool new: location type / Herramienta nueva: tipo de puesto
   // // MTIF[6].LocType : Werkzeug neu: Platzart / Tool new: location type / Herramienta nueva: tipo de puesto
   // // MTIF[7].LocType : Werkzeug neu: Platzart / Tool new: location type / Herramienta nueva: tipo de puesto
   // // MTIF[8].LocType : Werkzeug neu: Platzart / Tool new: location type / Herramienta nueva: tipo de puesto
   // // MTIF[9].LocType : Werkzeug neu: Platzart / Tool new: location type / Herramienta nueva: tipo de puesto
   // // MTIF[10].LocType : Werkzeug neu: Platzart / Tool new: location type / Herramienta nueva: tipo de puesto
   // // MTIF[11].LocType : Werkzeug neu: Platzart / Tool new: location type / Herramienta nueva: tipo de puesto
   // // MTIF[12].LocType : Werkzeug neu: Platzart / Tool new: location type / Herramienta nueva: tipo de puesto
   // // MTIF[13].LocType : Werkzeug neu: Platzart / Tool new: location type / Herramienta nueva: tipo de puesto
   // // MTIF[14].LocType : Werkzeug neu: Platzart / Tool new: location type / Herramienta nueva: tipo de puesto
   // // MTIF[15].LocType : Werkzeug neu: Platzart / Tool new: location type / Herramienta nueva: tipo de puesto
   // // MTIF[16].LocType : Werkzeug neu: Platzart / Tool new: location type / Herramienta nueva: tipo de puesto
   // // MTIF[2].SLeft : Werkeug neu: Größe links / Tool new: size left / Herramienta nueva: tamaño izquierda
   // // MTIF[3].SLeft : Werkeug neu: Größe links / Tool new: size left / Herramienta nueva: tamaño izquierda
   // // MTIF[4].SLeft : Werkeug neu: Größe links / Tool new: size left / Herramienta nueva: tamaño izquierda
   // // MTIF[5].SLeft : Werkeug neu: Größe links / Tool new: size left / Herramienta nueva: tamaño izquierda
   // // MTIF[6].SLeft : Werkeug neu: Größe links / Tool new: size left / Herramienta nueva: tamaño izquierda
   // // MTIF[7].SLeft : Werkeug neu: Größe links / Tool new: size left / Herramienta nueva: tamaño izquierda
   // // MTIF[8].SLeft : Werkeug neu: Größe links / Tool new: size left / Herramienta nueva: tamaño izquierda
   // // MTIF[9].SLeft : Werkeug neu: Größe links / Tool new: size left / Herramienta nueva: tamaño izquierda
   // // MTIF[10].SLeft : Werkeug neu: Größe links / Tool new: size left / Herramienta nueva: tamaño izquierda
   // // MTIF[11].SLeft : Werkeug neu: Größe links / Tool new: size left / Herramienta nueva: tamaño izquierda
   // // MTIF[12].SLeft : Werkeug neu: Größe links / Tool new: size left / Herramienta nueva: tamaño izquierda
   // // MTIF[13].SLeft : Werkeug neu: Größe links / Tool new: size left / Herramienta nueva: tamaño izquierda
   // // MTIF[14].SLeft : Werkeug neu: Größe links / Tool new: size left / Herramienta nueva: tamaño izquierda
   // // MTIF[15].SLeft : Werkeug neu: Größe links / Tool new: size left / Herramienta nueva: tamaño izquierda
   // // MTIF[16].SLeft : Werkeug neu: Größe links / Tool new: size left / Herramienta nueva: tamaño izquierda
   // // MTIF[2].SRight : Werkeug neu: Größe rechts / Tool new: size right / Herramienta nueva: tamaño derecha
   // // MTIF[3].SRight : Werkeug neu: Größe rechts / Tool new: size right / Herramienta nueva: tamaño derecha
   // // MTIF[4].SRight : Werkeug neu: Größe rechts / Tool new: size right / Herramienta nueva: tamaño derecha
   // // MTIF[5].SRight : Werkeug neu: Größe rechts / Tool new: size right / Herramienta nueva: tamaño derecha
   // // MTIF[6].SRight : Werkeug neu: Größe rechts / Tool new: size right / Herramienta nueva: tamaño derecha
   // // MTIF[7].SRight : Werkeug neu: Größe rechts / Tool new: size right / Herramienta nueva: tamaño derecha
   // // MTIF[8].SRight : Werkeug neu: Größe rechts / Tool new: size right / Herramienta nueva: tamaño derecha
   // // MTIF[9].SRight : Werkeug neu: Größe rechts / Tool new: size right / Herramienta nueva: tamaño derecha
   // // MTIF[10].SRight : Werkeug neu: Größe rechts / Tool new: size right / Herramienta nueva: tamaño derecha
   // // MTIF[11].SRight : Werkeug neu: Größe rechts / Tool new: size right / Herramienta nueva: tamaño derecha
   // // MTIF[12].SRight : Werkeug neu: Größe rechts / Tool new: size right / Herramienta nueva: tamaño derecha
   // // MTIF[13].SRight : Werkeug neu: Größe rechts / Tool new: size right / Herramienta nueva: tamaño derecha
   // // MTIF[14].SRight : Werkeug neu: Größe rechts / Tool new: size right / Herramienta nueva: tamaño derecha
   // // MTIF[15].SRight : Werkeug neu: Größe rechts / Tool new: size right / Herramienta nueva: tamaño derecha
   // // MTIF[16].SRight : Werkeug neu: Größe rechts / Tool new: size right / Herramienta nueva: tamaño derecha
   // // MTIF[2].STop : Werkeug neu: Größe oben / Tool new: size top / Herramienta nueva: tamaño arriba
   // // MTIF[3].STop : Werkeug neu: Größe oben / Tool new: size top / Herramienta nueva: tamaño arriba
   // // MTIF[4].STop : Werkeug neu: Größe oben / Tool new: size top / Herramienta nueva: tamaño arriba
   // // MTIF[5].STop : Werkeug neu: Größe oben / Tool new: size top / Herramienta nueva: tamaño arriba
   // // MTIF[6].STop : Werkeug neu: Größe oben / Tool new: size top / Herramienta nueva: tamaño arriba
   // // MTIF[7].STop : Werkeug neu: Größe oben / Tool new: size top / Herramienta nueva: tamaño arriba
   // // MTIF[8].STop : Werkeug neu: Größe oben / Tool new: size top / Herramienta nueva: tamaño arriba
   // // MTIF[9].STop : Werkeug neu: Größe oben / Tool new: size top / Herramienta nueva: tamaño arriba
   // // MTIF[10].STop : Werkeug neu: Größe oben / Tool new: size top / Herramienta nueva: tamaño arriba
   // // MTIF[11].STop : Werkeug neu: Größe oben / Tool new: size top / Herramienta nueva: tamaño arriba
   // // MTIF[12].STop : Werkeug neu: Größe oben / Tool new: size top / Herramienta nueva: tamaño arriba
   // // MTIF[13].STop : Werkeug neu: Größe oben / Tool new: size top / Herramienta nueva: tamaño arriba
   // // MTIF[14].STop : Werkeug neu: Größe oben / Tool new: size top / Herramienta nueva: tamaño arriba
   // // MTIF[15].STop : Werkeug neu: Größe oben / Tool new: size top / Herramienta nueva: tamaño arriba
   // // MTIF[16].STop : Werkeug neu: Größe oben / Tool new: size top / Herramienta nueva: tamaño arriba
   // // MTIF[2].SBottom : Werkeug neu: Größe unten / Tool new: size bottom / Herramienta nueva: tamaño abajo
   // // MTIF[3].SBottom : Werkeug neu: Größe unten / Tool new: size bottom / Herramienta nueva: tamaño abajo
   // // MTIF[4].SBottom : Werkeug neu: Größe unten / Tool new: size bottom / Herramienta nueva: tamaño abajo
   // // MTIF[5].SBottom : Werkeug neu: Größe unten / Tool new: size bottom / Herramienta nueva: tamaño abajo
   // // MTIF[6].SBottom : Werkeug neu: Größe unten / Tool new: size bottom / Herramienta nueva: tamaño abajo
   // // MTIF[7].SBottom : Werkeug neu: Größe unten / Tool new: size bottom / Herramienta nueva: tamaño abajo
   // // MTIF[8].SBottom : Werkeug neu: Größe unten / Tool new: size bottom / Herramienta nueva: tamaño abajo
   // // MTIF[9].SBottom : Werkeug neu: Größe unten / Tool new: size bottom / Herramienta nueva: tamaño abajo
   // // MTIF[10].SBottom : Werkeug neu: Größe unten / Tool new: size bottom / Herramienta nueva: tamaño abajo
   // // MTIF[11].SBottom : Werkeug neu: Größe unten / Tool new: size bottom / Herramienta nueva: tamaño abajo
   // // MTIF[12].SBottom : Werkeug neu: Größe unten / Tool new: size bottom / Herramienta nueva: tamaño abajo
   // // MTIF[13].SBottom : Werkeug neu: Größe unten / Tool new: size bottom / Herramienta nueva: tamaño abajo
   // // MTIF[14].SBottom : Werkeug neu: Größe unten / Tool new: size bottom / Herramienta nueva: tamaño abajo
   // // MTIF[15].SBottom : Werkeug neu: Größe unten / Tool new: size bottom / Herramienta nueva: tamaño abajo
   // // MTIF[16].SBottom : Werkeug neu: Größe unten / Tool new: size bottom / Herramienta nueva: tamaño abajo
   // // MTIF[2].TInBuffer : ID für Werkzeuge im Puffer / ID for tools in buffer / ID para herramientas en búfer
   // // MTIF[3].TInBuffer : ID für Werkzeuge im Puffer / ID for tools in buffer / ID para herramientas en búfer
   // // MTIF[4].TInBuffer : ID für Werkzeuge im Puffer / ID for tools in buffer / ID para herramientas en búfer
   // // MTIF[5].TInBuffer : ID für Werkzeuge im Puffer / ID for tools in buffer / ID para herramientas en búfer
   // // MTIF[6].TInBuffer : ID für Werkzeuge im Puffer / ID for tools in buffer / ID para herramientas en búfer
   // // MTIF[7].TInBuffer : ID für Werkzeuge im Puffer / ID for tools in buffer / ID para herramientas en búfer
   // // MTIF[8].TInBuffer : ID für Werkzeuge im Puffer / ID for tools in buffer / ID para herramientas en búfer
   // // MTIF[9].TInBuffer : ID für Werkzeuge im Puffer / ID for tools in buffer / ID para herramientas en búfer
   // // MTIF[10].TInBuffer : ID für Werkzeuge im Puffer / ID for tools in buffer / ID para herramientas en búfer
   // // MTIF[11].TInBuffer : ID für Werkzeuge im Puffer / ID for tools in buffer / ID para herramientas en búfer
   // // MTIF[12].TInBuffer : ID für Werkzeuge im Puffer / ID for tools in buffer / ID para herramientas en búfer
   // // MTIF[13].TInBuffer : ID für Werkzeuge im Puffer / ID for tools in buffer / ID para herramientas en búfer
   // // MTIF[14].TInBuffer : ID für Werkzeuge im Puffer / ID for tools in buffer / ID para herramientas en búfer
   // // MTIF[15].TInBuffer : ID für Werkzeuge im Puffer / ID for tools in buffer / ID para herramientas en búfer
   // // MTIF[16].TInBuffer : ID für Werkzeuge im Puffer / ID for tools in buffer / ID para herramientas en búfer
   // // MTIF[2].IgnoreDisabled : Deaktiviert ignorieren / Ignore disabled / Ignorar desactivado
   // // MTIF[3].IgnoreDisabled : Deaktiviert ignorieren / Ignore disabled / Ignorar desactivado
   // // MTIF[4].IgnoreDisabled : Deaktiviert ignorieren / Ignore disabled / Ignorar desactivado
   // // MTIF[5].IgnoreDisabled : Deaktiviert ignorieren / Ignore disabled / Ignorar desactivado
   // // MTIF[6].IgnoreDisabled : Deaktiviert ignorieren / Ignore disabled / Ignorar desactivado
   // // MTIF[7].IgnoreDisabled : Deaktiviert ignorieren / Ignore disabled / Ignorar desactivado
   // // MTIF[8].IgnoreDisabled : Deaktiviert ignorieren / Ignore disabled / Ignorar desactivado
   // // MTIF[9].IgnoreDisabled : Deaktiviert ignorieren / Ignore disabled / Ignorar desactivado
   // // MTIF[10].IgnoreDisabled : Deaktiviert ignorieren / Ignore disabled / Ignorar desactivado
   // // MTIF[11].IgnoreDisabled : Deaktiviert ignorieren / Ignore disabled / Ignorar desactivado
   // // MTIF[12].IgnoreDisabled : Deaktiviert ignorieren / Ignore disabled / Ignorar desactivado
   // // MTIF[13].IgnoreDisabled : Deaktiviert ignorieren / Ignore disabled / Ignorar desactivado
   // // MTIF[14].IgnoreDisabled : Deaktiviert ignorieren / Ignore disabled / Ignorar desactivado
   // // MTIF[15].IgnoreDisabled : Deaktiviert ignorieren / Ignore disabled / Ignorar desactivado
   // // MTIF[16].IgnoreDisabled : Deaktiviert ignorieren / Ignore disabled / Ignorar desactivado
   // // MTIF[2].Unload : Zu entladen / To be unloaded / Por descargar
   // // MTIF[3].Unload : Zu entladen / To be unloaded / Por descargar
   // // MTIF[4].Unload : Zu entladen / To be unloaded / Por descargar
   // // MTIF[5].Unload : Zu entladen / To be unloaded / Por descargar
   // // MTIF[6].Unload : Zu entladen / To be unloaded / Por descargar
   // // MTIF[7].Unload : Zu entladen / To be unloaded / Por descargar
   // // MTIF[8].Unload : Zu entladen / To be unloaded / Por descargar
   // // MTIF[9].Unload : Zu entladen / To be unloaded / Por descargar
   // // MTIF[10].Unload : Zu entladen / To be unloaded / Por descargar
   // // MTIF[11].Unload : Zu entladen / To be unloaded / Por descargar
   // // MTIF[12].Unload : Zu entladen / To be unloaded / Por descargar
   // // MTIF[13].Unload : Zu entladen / To be unloaded / Por descargar
   // // MTIF[14].Unload : Zu entladen / To be unloaded / Por descargar
   // // MTIF[15].Unload : Zu entladen / To be unloaded / Por descargar
   // // MTIF[16].Unload : Zu entladen / To be unloaded / Por descargar
   // // MTIF[2].Load : Zu laden / To be loaded / Por cargar
   // // MTIF[3].Load : Zu laden / To be loaded / Por cargar
   // // MTIF[4].Load : Zu laden / To be loaded / Por cargar
   // // MTIF[5].Load : Zu laden / To be loaded / Por cargar
   // // MTIF[6].Load : Zu laden / To be loaded / Por cargar
   // // MTIF[7].Load : Zu laden / To be loaded / Por cargar
   // // MTIF[8].Load : Zu laden / To be loaded / Por cargar
   // // MTIF[9].Load : Zu laden / To be loaded / Por cargar
   // // MTIF[10].Load : Zu laden / To be loaded / Por cargar
   // // MTIF[11].Load : Zu laden / To be loaded / Por cargar
   // // MTIF[12].Load : Zu laden / To be loaded / Por cargar
   // // MTIF[13].Load : Zu laden / To be loaded / Por cargar
   // // MTIF[14].Load : Zu laden / To be loaded / Por cargar
   // // MTIF[15].Load : Zu laden / To be loaded / Por cargar
   // // MTIF[16].Load : Zu laden / To be loaded / Por cargar
   // // MTIF[2].MasterTool : Master-Werkzeug / Master tool / Herramienta maestra
   // // MTIF[3].MasterTool : Master-Werkzeug / Master tool / Herramienta maestra
   // // MTIF[4].MasterTool : Master-Werkzeug / Master tool / Herramienta maestra
   // // MTIF[5].MasterTool : Master-Werkzeug / Master tool / Herramienta maestra
   // // MTIF[6].MasterTool : Master-Werkzeug / Master tool / Herramienta maestra
   // // MTIF[7].MasterTool : Master-Werkzeug / Master tool / Herramienta maestra
   // // MTIF[8].MasterTool : Master-Werkzeug / Master tool / Herramienta maestra
   // // MTIF[9].MasterTool : Master-Werkzeug / Master tool / Herramienta maestra
   // // MTIF[10].MasterTool : Master-Werkzeug / Master tool / Herramienta maestra
   // // MTIF[11].MasterTool : Master-Werkzeug / Master tool / Herramienta maestra
   // // MTIF[12].MasterTool : Master-Werkzeug / Master tool / Herramienta maestra
   // // MTIF[13].MasterTool : Master-Werkzeug / Master tool / Herramienta maestra
   // // MTIF[14].MasterTool : Master-Werkzeug / Master tool / Herramienta maestra
   // // MTIF[15].MasterTool : Master-Werkzeug / Master tool / Herramienta maestra
   // // MTIF[16].MasterTool : Master-Werkzeug / Master tool / Herramienta maestra
   // // MTIF[2].n26_5 : Reserviert / Reserved / Reservado
   // // MTIF[3].n26_5 : Reserviert / Reserved / Reservado
   // // MTIF[4].n26_5 : Reserviert / Reserved / Reservado
   // // MTIF[5].n26_5 : Reserviert / Reserved / Reservado
   // // MTIF[6].n26_5 : Reserviert / Reserved / Reservado
   // // MTIF[7].n26_5 : Reserviert / Reserved / Reservado
   // // MTIF[8].n26_5 : Reserviert / Reserved / Reservado
   // // MTIF[9].n26_5 : Reserviert / Reserved / Reservado
   // // MTIF[10].n26_5 : Reserviert / Reserved / Reservado
   // // MTIF[11].n26_5 : Reserviert / Reserved / Reservado
   // // MTIF[12].n26_5 : Reserviert / Reserved / Reservado
   // // MTIF[13].n26_5 : Reserviert / Reserved / Reservado
   // // MTIF[14].n26_5 : Reserviert / Reserved / Reservado
   // // MTIF[15].n26_5 : Reserviert / Reserved / Reservado
   // // MTIF[16].n26_5 : Reserviert / Reserved / Reservado
   // // MTIF[2].n26_6 : Reserviert / Reserved / Reservado
   // // MTIF[3].n26_6 : Reserviert / Reserved / Reservado
   // // MTIF[4].n26_6 : Reserviert / Reserved / Reservado
   // // MTIF[5].n26_6 : Reserviert / Reserved / Reservado
   // // MTIF[6].n26_6 : Reserviert / Reserved / Reservado
   // // MTIF[7].n26_6 : Reserviert / Reserved / Reservado
   // // MTIF[8].n26_6 : Reserviert / Reserved / Reservado
   // // MTIF[9].n26_6 : Reserviert / Reserved / Reservado
   // // MTIF[10].n26_6 : Reserviert / Reserved / Reservado
   // // MTIF[11].n26_6 : Reserviert / Reserved / Reservado
   // // MTIF[12].n26_6 : Reserviert / Reserved / Reservado
   // // MTIF[13].n26_6 : Reserviert / Reserved / Reservado
   // // MTIF[14].n26_6 : Reserviert / Reserved / Reservado
   // // MTIF[15].n26_6 : Reserviert / Reserved / Reservado
   // // MTIF[16].n26_6 : Reserviert / Reserved / Reservado
   // // MTIF[2].HandTool : Handwerkzeug / Hand tool / Herramienta manual
   // // MTIF[3].HandTool : Handwerkzeug / Hand tool / Herramienta manual
   // // MTIF[4].HandTool : Handwerkzeug / Hand tool / Herramienta manual
   // // MTIF[5].HandTool : Handwerkzeug / Hand tool / Herramienta manual
   // // MTIF[6].HandTool : Handwerkzeug / Hand tool / Herramienta manual
   // // MTIF[7].HandTool : Handwerkzeug / Hand tool / Herramienta manual
   // // MTIF[8].HandTool : Handwerkzeug / Hand tool / Herramienta manual
   // // MTIF[9].HandTool : Handwerkzeug / Hand tool / Herramienta manual
   // // MTIF[10].HandTool : Handwerkzeug / Hand tool / Herramienta manual
   // // MTIF[11].HandTool : Handwerkzeug / Hand tool / Herramienta manual
   // // MTIF[12].HandTool : Handwerkzeug / Hand tool / Herramienta manual
   // // MTIF[13].HandTool : Handwerkzeug / Hand tool / Herramienta manual
   // // MTIF[14].HandTool : Handwerkzeug / Hand tool / Herramienta manual
   // // MTIF[15].HandTool : Handwerkzeug / Hand tool / Herramienta manual
   // // MTIF[16].HandTool : Handwerkzeug / Hand tool / Herramienta manual
   // // MTIF[2].Active : Aktives Werkzeug / Active tool / Herramienta activa
   // // MTIF[3].Active : Aktives Werkzeug / Active tool / Herramienta activa
   // // MTIF[4].Active : Aktives Werkzeug / Active tool / Herramienta activa
   // // MTIF[5].Active : Aktives Werkzeug / Active tool / Herramienta activa
   // // MTIF[6].Active : Aktives Werkzeug / Active tool / Herramienta activa
   // // MTIF[7].Active : Aktives Werkzeug / Active tool / Herramienta activa
   // // MTIF[8].Active : Aktives Werkzeug / Active tool / Herramienta activa
   // // MTIF[9].Active : Aktives Werkzeug / Active tool / Herramienta activa
   // // MTIF[10].Active : Aktives Werkzeug / Active tool / Herramienta activa
   // // MTIF[11].Active : Aktives Werkzeug / Active tool / Herramienta activa
   // // MTIF[12].Active : Aktives Werkzeug / Active tool / Herramienta activa
   // // MTIF[13].Active : Aktives Werkzeug / Active tool / Herramienta activa
   // // MTIF[14].Active : Aktives Werkzeug / Active tool / Herramienta activa
   // // MTIF[15].Active : Aktives Werkzeug / Active tool / Herramienta activa
   // // MTIF[16].Active : Aktives Werkzeug / Active tool / Herramienta activa
   // // MTIF[2].Enabled : Werkzeug aktiviert / Tool enabled / Herramienta activada
   // // MTIF[3].Enabled : Werkzeug aktiviert / Tool enabled / Herramienta activada
   // // MTIF[4].Enabled : Werkzeug aktiviert / Tool enabled / Herramienta activada
   // // MTIF[5].Enabled : Werkzeug aktiviert / Tool enabled / Herramienta activada
   // // MTIF[6].Enabled : Werkzeug aktiviert / Tool enabled / Herramienta activada
   // // MTIF[7].Enabled : Werkzeug aktiviert / Tool enabled / Herramienta activada
   // // MTIF[8].Enabled : Werkzeug aktiviert / Tool enabled / Herramienta activada
   // // MTIF[9].Enabled : Werkzeug aktiviert / Tool enabled / Herramienta activada
   // // MTIF[10].Enabled : Werkzeug aktiviert / Tool enabled / Herramienta activada
   // // MTIF[11].Enabled : Werkzeug aktiviert / Tool enabled / Herramienta activada
   // // MTIF[12].Enabled : Werkzeug aktiviert / Tool enabled / Herramienta activada
   // // MTIF[13].Enabled : Werkzeug aktiviert / Tool enabled / Herramienta activada
   // // MTIF[14].Enabled : Werkzeug aktiviert / Tool enabled / Herramienta activada
   // // MTIF[15].Enabled : Werkzeug aktiviert / Tool enabled / Herramienta activada
   // // MTIF[16].Enabled : Werkzeug aktiviert / Tool enabled / Herramienta activada
   // // MTIF[2].Disabled : Werkzeug deaktiviert / Tool disabled / Herramienta desactivada
   // // MTIF[3].Disabled : Werkzeug deaktiviert / Tool disabled / Herramienta desactivada
   // // MTIF[4].Disabled : Werkzeug deaktiviert / Tool disabled / Herramienta desactivada
   // // MTIF[5].Disabled : Werkzeug deaktiviert / Tool disabled / Herramienta desactivada
   // // MTIF[6].Disabled : Werkzeug deaktiviert / Tool disabled / Herramienta desactivada
   // // MTIF[7].Disabled : Werkzeug deaktiviert / Tool disabled / Herramienta desactivada
   // // MTIF[8].Disabled : Werkzeug deaktiviert / Tool disabled / Herramienta desactivada
   // // MTIF[9].Disabled : Werkzeug deaktiviert / Tool disabled / Herramienta desactivada
   // // MTIF[10].Disabled : Werkzeug deaktiviert / Tool disabled / Herramienta desactivada
   // // MTIF[11].Disabled : Werkzeug deaktiviert / Tool disabled / Herramienta desactivada
   // // MTIF[12].Disabled : Werkzeug deaktiviert / Tool disabled / Herramienta desactivada
   // // MTIF[13].Disabled : Werkzeug deaktiviert / Tool disabled / Herramienta desactivada
   // // MTIF[14].Disabled : Werkzeug deaktiviert / Tool disabled / Herramienta desactivada
   // // MTIF[15].Disabled : Werkzeug deaktiviert / Tool disabled / Herramienta desactivada
   // // MTIF[16].Disabled : Werkzeug deaktiviert / Tool disabled / Herramienta desactivada
   // // MTIF[2].Measured : Werkzeug gemessen / Tool measured / Herramienta medida
   // // MTIF[3].Measured : Werkzeug gemessen / Tool measured / Herramienta medida
   // // MTIF[4].Measured : Werkzeug gemessen / Tool measured / Herramienta medida
   // // MTIF[5].Measured : Werkzeug gemessen / Tool measured / Herramienta medida
   // // MTIF[6].Measured : Werkzeug gemessen / Tool measured / Herramienta medida
   // // MTIF[7].Measured : Werkzeug gemessen / Tool measured / Herramienta medida
   // // MTIF[8].Measured : Werkzeug gemessen / Tool measured / Herramienta medida
   // // MTIF[9].Measured : Werkzeug gemessen / Tool measured / Herramienta medida
   // // MTIF[10].Measured : Werkzeug gemessen / Tool measured / Herramienta medida
   // // MTIF[11].Measured : Werkzeug gemessen / Tool measured / Herramienta medida
   // // MTIF[12].Measured : Werkzeug gemessen / Tool measured / Herramienta medida
   // // MTIF[13].Measured : Werkzeug gemessen / Tool measured / Herramienta medida
   // // MTIF[14].Measured : Werkzeug gemessen / Tool measured / Herramienta medida
   // // MTIF[15].Measured : Werkzeug gemessen / Tool measured / Herramienta medida
   // // MTIF[16].Measured : Werkzeug gemessen / Tool measured / Herramienta medida
   // // MTIF[2].Prewarn : Vorwarnungsgrenze erreicht / Prewarning limit reached / Límite de prealarma alcanzado
   // // MTIF[3].Prewarn : Vorwarnungsgrenze erreicht / Prewarning limit reached / Límite de prealarma alcanzado
   // // MTIF[4].Prewarn : Vorwarnungsgrenze erreicht / Prewarning limit reached / Límite de prealarma alcanzado
   // // MTIF[5].Prewarn : Vorwarnungsgrenze erreicht / Prewarning limit reached / Límite de prealarma alcanzado
   // // MTIF[6].Prewarn : Vorwarnungsgrenze erreicht / Prewarning limit reached / Límite de prealarma alcanzado
   // // MTIF[7].Prewarn : Vorwarnungsgrenze erreicht / Prewarning limit reached / Límite de prealarma alcanzado
   // // MTIF[8].Prewarn : Vorwarnungsgrenze erreicht / Prewarning limit reached / Límite de prealarma alcanzado
   // // MTIF[9].Prewarn : Vorwarnungsgrenze erreicht / Prewarning limit reached / Límite de prealarma alcanzado
   // // MTIF[10].Prewarn : Vorwarnungsgrenze erreicht / Prewarning limit reached / Límite de prealarma alcanzado
   // // MTIF[11].Prewarn : Vorwarnungsgrenze erreicht / Prewarning limit reached / Límite de prealarma alcanzado
   // // MTIF[12].Prewarn : Vorwarnungsgrenze erreicht / Prewarning limit reached / Límite de prealarma alcanzado
   // // MTIF[13].Prewarn : Vorwarnungsgrenze erreicht / Prewarning limit reached / Límite de prealarma alcanzado
   // // MTIF[14].Prewarn : Vorwarnungsgrenze erreicht / Prewarning limit reached / Límite de prealarma alcanzado
   // // MTIF[15].Prewarn : Vorwarnungsgrenze erreicht / Prewarning limit reached / Límite de prealarma alcanzado
   // // MTIF[16].Prewarn : Vorwarnungsgrenze erreicht / Prewarning limit reached / Límite de prealarma alcanzado
   // // MTIF[2].Change : Werkzeug wird gewechselt / Tool being changed / Sustituyendo herramienta
   // // MTIF[3].Change : Werkzeug wird gewechselt / Tool being changed / Sustituyendo herramienta
   // // MTIF[4].Change : Werkzeug wird gewechselt / Tool being changed / Sustituyendo herramienta
   // // MTIF[5].Change : Werkzeug wird gewechselt / Tool being changed / Sustituyendo herramienta
   // // MTIF[6].Change : Werkzeug wird gewechselt / Tool being changed / Sustituyendo herramienta
   // // MTIF[7].Change : Werkzeug wird gewechselt / Tool being changed / Sustituyendo herramienta
   // // MTIF[8].Change : Werkzeug wird gewechselt / Tool being changed / Sustituyendo herramienta
   // // MTIF[9].Change : Werkzeug wird gewechselt / Tool being changed / Sustituyendo herramienta
   // // MTIF[10].Change : Werkzeug wird gewechselt / Tool being changed / Sustituyendo herramienta
   // // MTIF[11].Change : Werkzeug wird gewechselt / Tool being changed / Sustituyendo herramienta
   // // MTIF[12].Change : Werkzeug wird gewechselt / Tool being changed / Sustituyendo herramienta
   // // MTIF[13].Change : Werkzeug wird gewechselt / Tool being changed / Sustituyendo herramienta
   // // MTIF[14].Change : Werkzeug wird gewechselt / Tool being changed / Sustituyendo herramienta
   // // MTIF[15].Change : Werkzeug wird gewechselt / Tool being changed / Sustituyendo herramienta
   // // MTIF[16].Change : Werkzeug wird gewechselt / Tool being changed / Sustituyendo herramienta
   // // MTIF[2].FixedLoc : Werkzeug-Festplatz codiert / Tool fixed location coded / Puesto fijo de herramienta codificado
   // // MTIF[3].FixedLoc : Werkzeug-Festplatz codiert / Tool fixed location coded / Puesto fijo de herramienta codificado
   // // MTIF[4].FixedLoc : Werkzeug-Festplatz codiert / Tool fixed location coded / Puesto fijo de herramienta codificado
   // // MTIF[5].FixedLoc : Werkzeug-Festplatz codiert / Tool fixed location coded / Puesto fijo de herramienta codificado
   // // MTIF[6].FixedLoc : Werkzeug-Festplatz codiert / Tool fixed location coded / Puesto fijo de herramienta codificado
   // // MTIF[7].FixedLoc : Werkzeug-Festplatz codiert / Tool fixed location coded / Puesto fijo de herramienta codificado
   // // MTIF[8].FixedLoc : Werkzeug-Festplatz codiert / Tool fixed location coded / Puesto fijo de herramienta codificado
   // // MTIF[9].FixedLoc : Werkzeug-Festplatz codiert / Tool fixed location coded / Puesto fijo de herramienta codificado
   // // MTIF[10].FixedLoc : Werkzeug-Festplatz codiert / Tool fixed location coded / Puesto fijo de herramienta codificado
   // // MTIF[11].FixedLoc : Werkzeug-Festplatz codiert / Tool fixed location coded / Puesto fijo de herramienta codificado
   // // MTIF[12].FixedLoc : Werkzeug-Festplatz codiert / Tool fixed location coded / Puesto fijo de herramienta codificado
   // // MTIF[13].FixedLoc : Werkzeug-Festplatz codiert / Tool fixed location coded / Puesto fijo de herramienta codificado
   // // MTIF[14].FixedLoc : Werkzeug-Festplatz codiert / Tool fixed location coded / Puesto fijo de herramienta codificado
   // // MTIF[15].FixedLoc : Werkzeug-Festplatz codiert / Tool fixed location coded / Puesto fijo de herramienta codificado
   // // MTIF[16].FixedLoc : Werkzeug-Festplatz codiert / Tool fixed location coded / Puesto fijo de herramienta codificado
   // // MTIF[2].Used : Werkzeug war in Gebrauch / Tool was in use / La herramienta estaba en uso
   // // MTIF[3].Used : Werkzeug war in Gebrauch / Tool was in use / La herramienta estaba en uso
   // // MTIF[4].Used : Werkzeug war in Gebrauch / Tool was in use / La herramienta estaba en uso
   // // MTIF[5].Used : Werkzeug war in Gebrauch / Tool was in use / La herramienta estaba en uso
   // // MTIF[6].Used : Werkzeug war in Gebrauch / Tool was in use / La herramienta estaba en uso
   // // MTIF[7].Used : Werkzeug war in Gebrauch / Tool was in use / La herramienta estaba en uso
   // // MTIF[8].Used : Werkzeug war in Gebrauch / Tool was in use / La herramienta estaba en uso
   // // MTIF[9].Used : Werkzeug war in Gebrauch / Tool was in use / La herramienta estaba en uso
   // // MTIF[10].Used : Werkzeug war in Gebrauch / Tool was in use / La herramienta estaba en uso
   // // MTIF[11].Used : Werkzeug war in Gebrauch / Tool was in use / La herramienta estaba en uso
   // // MTIF[12].Used : Werkzeug war in Gebrauch / Tool was in use / La herramienta estaba en uso
   // // MTIF[13].Used : Werkzeug war in Gebrauch / Tool was in use / La herramienta estaba en uso
   // // MTIF[14].Used : Werkzeug war in Gebrauch / Tool was in use / La herramienta estaba en uso
   // // MTIF[15].Used : Werkzeug war in Gebrauch / Tool was in use / La herramienta estaba en uso
   // // MTIF[16].Used : Werkzeug war in Gebrauch / Tool was in use / La herramienta estaba en uso
   // // MTIF[2].TNo : Werkzeug neu: WZ-Nummer / Tool new: T number / Herramienta nueva: n.º herramienta
   // // MTIF[3].TNo : Werkzeug neu: WZ-Nummer / Tool new: T number / Herramienta nueva: n.º herramienta
   // // MTIF[4].TNo : Werkzeug neu: WZ-Nummer / Tool new: T number / Herramienta nueva: n.º herramienta
   // // MTIF[5].TNo : Werkzeug neu: WZ-Nummer / Tool new: T number / Herramienta nueva: n.º herramienta
   // // MTIF[6].TNo : Werkzeug neu: WZ-Nummer / Tool new: T number / Herramienta nueva: n.º herramienta
   // // MTIF[7].TNo : Werkzeug neu: WZ-Nummer / Tool new: T number / Herramienta nueva: n.º herramienta
   // // MTIF[8].TNo : Werkzeug neu: WZ-Nummer / Tool new: T number / Herramienta nueva: n.º herramienta
   // // MTIF[9].TNo : Werkzeug neu: WZ-Nummer / Tool new: T number / Herramienta nueva: n.º herramienta
   // // MTIF[10].TNo : Werkzeug neu: WZ-Nummer / Tool new: T number / Herramienta nueva: n.º herramienta
   // // MTIF[11].TNo : Werkzeug neu: WZ-Nummer / Tool new: T number / Herramienta nueva: n.º herramienta
   // // MTIF[12].TNo : Werkzeug neu: WZ-Nummer / Tool new: T number / Herramienta nueva: n.º herramienta
   // // MTIF[13].TNo : Werkzeug neu: WZ-Nummer / Tool new: T number / Herramienta nueva: n.º herramienta
   // // MTIF[14].TNo : Werkzeug neu: WZ-Nummer / Tool new: T number / Herramienta nueva: n.º herramienta
   // // MTIF[15].TNo : Werkzeug neu: WZ-Nummer / Tool new: T number / Herramienta nueva: n.º herramienta
   // // MTIF[16].TNo : Werkzeug neu: WZ-Nummer / Tool new: T number / Herramienta nueva: n.º herramienta
   // // MTIF[2].Toolholder : Werkzeughalter-Nummer als Referenz für die Werkzeugkompensation / Toolholder number as tool compensation reference / Número de portaherramientas como referencia para compensación de herramientas
   // // MTIF[3].Toolholder : Werkzeughalter-Nummer als Referenz für die Werkzeugkompensation / Toolholder number as tool compensation reference / Número de portaherramientas como referencia para compensación de herramientas
   // // MTIF[4].Toolholder : Werkzeughalter-Nummer als Referenz für die Werkzeugkompensation / Toolholder number as tool compensation reference / Número de portaherramientas como referencia para compensación de herramientas
   // // MTIF[5].Toolholder : Werkzeughalter-Nummer als Referenz für die Werkzeugkompensation / Toolholder number as tool compensation reference / Número de portaherramientas como referencia para compensación de herramientas
   // // MTIF[6].Toolholder : Werkzeughalter-Nummer als Referenz für die Werkzeugkompensation / Toolholder number as tool compensation reference / Número de portaherramientas como referencia para compensación de herramientas
   // // MTIF[7].Toolholder : Werkzeughalter-Nummer als Referenz für die Werkzeugkompensation / Toolholder number as tool compensation reference / Número de portaherramientas como referencia para compensación de herramientas
   // // MTIF[8].Toolholder : Werkzeughalter-Nummer als Referenz für die Werkzeugkompensation / Toolholder number as tool compensation reference / Número de portaherramientas como referencia para compensación de herramientas
   // // MTIF[9].Toolholder : Werkzeughalter-Nummer als Referenz für die Werkzeugkompensation / Toolholder number as tool compensation reference / Número de portaherramientas como referencia para compensación de herramientas
   // // MTIF[10].Toolholder : Werkzeughalter-Nummer als Referenz für die Werkzeugkompensation / Toolholder number as tool compensation reference / Número de portaherramientas como referencia para compensación de herramientas
   // // MTIF[11].Toolholder : Werkzeughalter-Nummer als Referenz für die Werkzeugkompensation / Toolholder number as tool compensation reference / Número de portaherramientas como referencia para compensación de herramientas
   // // MTIF[12].Toolholder : Werkzeughalter-Nummer als Referenz für die Werkzeugkompensation / Toolholder number as tool compensation reference / Número de portaherramientas como referencia para compensación de herramientas
   // // MTIF[13].Toolholder : Werkzeughalter-Nummer als Referenz für die Werkzeugkompensation / Toolholder number as tool compensation reference / Número de portaherramientas como referencia para compensación de herramientas
   // // MTIF[14].Toolholder : Werkzeughalter-Nummer als Referenz für die Werkzeugkompensation / Toolholder number as tool compensation reference / Número de portaherramientas como referencia para compensación de herramientas
   // // MTIF[15].Toolholder : Werkzeughalter-Nummer als Referenz für die Werkzeugkompensation / Toolholder number as tool compensation reference / Número de portaherramientas como referencia para compensación de herramientas
   // // MTIF[16].Toolholder : Werkzeughalter-Nummer als Referenz für die Werkzeugkompensation / Toolholder number as tool compensation reference / Número de portaherramientas como referencia para compensación de herramientas
   // // MTIF[2].MyMag : Multitool-Nummer, in die das Werkzeug geladen wird / Multitool number the tool is loaded onto / Número de Multitool en el que se carga la herramienta
   // // MTIF[3].MyMag : Multitool-Nummer, in die das Werkzeug geladen wird / Multitool number the tool is loaded onto / Número de Multitool en el que se carga la herramienta
   // // MTIF[4].MyMag : Multitool-Nummer, in die das Werkzeug geladen wird / Multitool number the tool is loaded onto / Número de Multitool en el que se carga la herramienta
   // // MTIF[5].MyMag : Multitool-Nummer, in die das Werkzeug geladen wird / Multitool number the tool is loaded onto / Número de Multitool en el que se carga la herramienta
   // // MTIF[6].MyMag : Multitool-Nummer, in die das Werkzeug geladen wird / Multitool number the tool is loaded onto / Número de Multitool en el que se carga la herramienta
   // // MTIF[7].MyMag : Multitool-Nummer, in die das Werkzeug geladen wird / Multitool number the tool is loaded onto / Número de Multitool en el que se carga la herramienta
   // // MTIF[8].MyMag : Multitool-Nummer, in die das Werkzeug geladen wird / Multitool number the tool is loaded onto / Número de Multitool en el que se carga la herramienta
   // // MTIF[9].MyMag : Multitool-Nummer, in die das Werkzeug geladen wird / Multitool number the tool is loaded onto / Número de Multitool en el que se carga la herramienta
   // // MTIF[10].MyMag : Multitool-Nummer, in die das Werkzeug geladen wird / Multitool number the tool is loaded onto / Número de Multitool en el que se carga la herramienta
   // // MTIF[11].MyMag : Multitool-Nummer, in die das Werkzeug geladen wird / Multitool number the tool is loaded onto / Número de Multitool en el que se carga la herramienta
   // // MTIF[12].MyMag : Multitool-Nummer, in die das Werkzeug geladen wird / Multitool number the tool is loaded onto / Número de Multitool en el que se carga la herramienta
   // // MTIF[13].MyMag : Multitool-Nummer, in die das Werkzeug geladen wird / Multitool number the tool is loaded onto / Número de Multitool en el que se carga la herramienta
   // // MTIF[14].MyMag : Multitool-Nummer, in die das Werkzeug geladen wird / Multitool number the tool is loaded onto / Número de Multitool en el que se carga la herramienta
   // // MTIF[15].MyMag : Multitool-Nummer, in die das Werkzeug geladen wird / Multitool number the tool is loaded onto / Número de Multitool en el que se carga la herramienta
   // // MTIF[16].MyMag : Multitool-Nummer, in die das Werkzeug geladen wird / Multitool number the tool is loaded onto / Número de Multitool en el que se carga la herramienta
   // // MTIF[2].MyPlace : Multitool-Platznummer / Multitool place number / Número de puesto de Multitool
   // // MTIF[3].MyPlace : Multitool-Platznummer / Multitool place number / Número de puesto de Multitool
   // // MTIF[4].MyPlace : Multitool-Platznummer / Multitool place number / Número de puesto de Multitool
   // // MTIF[5].MyPlace : Multitool-Platznummer / Multitool place number / Número de puesto de Multitool
   // // MTIF[6].MyPlace : Multitool-Platznummer / Multitool place number / Número de puesto de Multitool
   // // MTIF[7].MyPlace : Multitool-Platznummer / Multitool place number / Número de puesto de Multitool
   // // MTIF[8].MyPlace : Multitool-Platznummer / Multitool place number / Número de puesto de Multitool
   // // MTIF[9].MyPlace : Multitool-Platznummer / Multitool place number / Número de puesto de Multitool
   // // MTIF[10].MyPlace : Multitool-Platznummer / Multitool place number / Número de puesto de Multitool
   // // MTIF[11].MyPlace : Multitool-Platznummer / Multitool place number / Número de puesto de Multitool
   // // MTIF[12].MyPlace : Multitool-Platznummer / Multitool place number / Número de puesto de Multitool
   // // MTIF[13].MyPlace : Multitool-Platznummer / Multitool place number / Número de puesto de Multitool
   // // MTIF[14].MyPlace : Multitool-Platznummer / Multitool place number / Número de puesto de Multitool
   // // MTIF[15].MyPlace : Multitool-Platznummer / Multitool place number / Número de puesto de Multitool
   // // MTIF[16].MyPlace : Multitool-Platznummer / Multitool place number / Número de puesto de Multitool
   // // MTIF[2].reserved : Reserviert / Reserved / Reservado
   // // MTIF[3].reserved : Reserviert / Reserved / Reservado
   // // MTIF[4].reserved : Reserviert / Reserved / Reservado
   // // MTIF[5].reserved : Reserviert / Reserved / Reservado
   // // MTIF[6].reserved : Reserviert / Reserved / Reservado
   // // MTIF[7].reserved : Reserviert / Reserved / Reservado
   // // MTIF[8].reserved : Reserviert / Reserved / Reservado
   // // MTIF[9].reserved : Reserviert / Reserved / Reservado
   // // MTIF[10].reserved : Reserviert / Reserved / Reservado
   // // MTIF[11].reserved : Reserviert / Reserved / Reservado
   // // MTIF[12].reserved : Reserviert / Reserved / Reservado
   // // MTIF[13].reserved : Reserviert / Reserved / Reservado
   // // MTIF[14].reserved : Reserviert / Reserved / Reservado
   // // MTIF[15].reserved : Reserviert / Reserved / Reservado
   // // MTIF[16].reserved : Reserviert / Reserved / Reservado
END_TYPE

